Staubli VAL3: back.pgx

public program back(string x_sItem)
  local num l_nValue
  local num l_nSize
begin
  // get the value
  call getPalletPos(x_sItem,l_nValue)
  call getSizePallet(x_sItem,l_nSize)
  // set the value -1
  if l_nValue>0
    call setPalletPos(x_sItem,l_nValue-1)
  else
    call setPalletPos(x_sItem,l_nSize-1)
  endIf
end
